// TIA Portal V18 export
FUNCTION_BLOCK "Aux_Motor_Control"   // FB12, LAD
{ S7_Optimized_Access := 'TRUE' }
// Written BY Kristopher Gimenez January 25,2023
// This block is used to control the Aux, and Cooler fan motors.
// stored: AutoNumber false, MemoryReserve 100, SetENOAutomatically false
   VAR
      AuxPumpStartTOF { S7_SetPoint := 'True'} : TOF_TIME;
      AuxPumpFailTON { S7_SetPoint := 'True'} : TON_TIME;
      CoolingFanFailTON { S7_SetPoint := 'True'} : TON_TIME;
      CoolingFanStartTON { S7_SetPoint := 'True'} : TOF_TIME;
   END_VAR
BEGIN

REGION Network 1: Aux Pump Start
   // TOFF used on Aux pump allows 2 seconds for functions to stop when system is disabled before pump is shutdown and to maintain while switching between Aux and TD Enabled
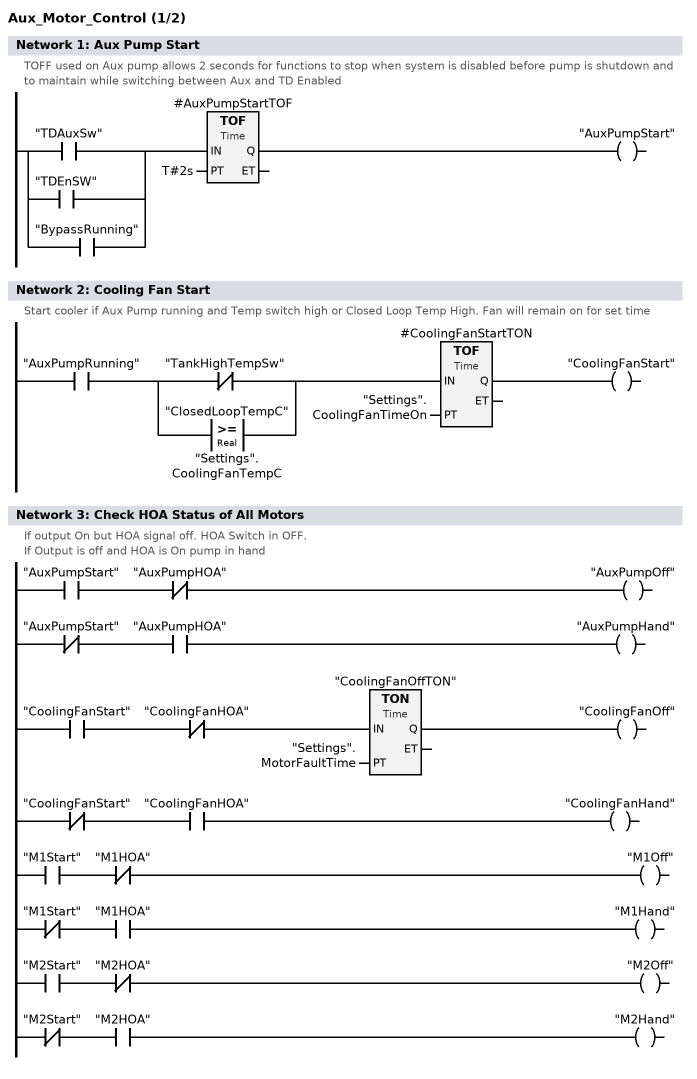
   RUNG wire#powerrail
      Contact( "TDAuxSw" )
      wire#w1
      { S7_Templates := "time_type := Time" } #AuxPumpStartTOF.TOF(pt := T#2s, et =>)
      Coil( "AuxPumpStart" )
   END_RUNG
   RUNG wire#powerrail
      Contact( "TDEnSW" )
   END_RUNG wire#w1
   RUNG wire#powerrail
      Contact( "BypassRunning" )
   END_RUNG wire#w1
   // the same network as SCL:
   #AuxPumpStartTOF(IN := "TDAuxSw" OR "TDEnSW" OR "BypassRunning", PT := T#2s);   // TOF
   "AuxPumpStart" := #AuxPumpStartTOF.Q;
END_REGION

REGION Network 2: Cooling Fan Start
   // Start cooler if Aux Pump running and Temp switch high or Closed Loop Temp High. Fan will remain on for set time
   RUNG wire#powerrail
      Contact( "AuxPumpRunning" )
      wire#w1
      I_Contact( "TankHighTempSw" )
      wire#w2
      { S7_Templates := "time_type := Time" } #CoolingFanStartTON.TOF(pt := "Settings".CoolingFanTimeOn, et =>)
      Coil( "CoolingFanStart" )
   END_RUNG
   RUNG wire#w1
      { S7_Templates := "SrcType := Real" } GE_Contact(in1 := "ClosedLoopTempC", in2 := "Settings".CoolingFanTempC)
   END_RUNG wire#w2
   // the same network as SCL:
   #CoolingFanStartTON(IN := "AuxPumpRunning" AND (NOT "TankHighTempSw" OR ("ClosedLoopTempC" >= "Settings".CoolingFanTempC)),   // TOF
                       PT := "Settings".CoolingFanTimeOn);
   "CoolingFanStart" := #CoolingFanStartTON.Q;
END_REGION

REGION Network 3: Check HOA Status of All Motors
   // If output On but HOA signal off. HOA Switch in OFF. 
   // If Output is off and HOA is On pump in hand
   RUNG wire#powerrail
      Contact( "AuxPumpStart" )
      I_Contact( "AuxPumpHOA" )
      Coil( "AuxPumpOff" )
   END_RUNG
   RUNG wire#powerrail
      I_Contact( "AuxPumpStart" )
      Contact( "AuxPumpHOA" )
      Coil( "AuxPumpHand" )
   END_RUNG
   RUNG wire#powerrail
      Contact( "CoolingFanStart" )
      I_Contact( "CoolingFanHOA" )
      { S7_Templates := "time_type := Time" } "CoolingFanOffTON".TON(pt := "Settings".MotorFaultTime, et =>)
      Coil( "CoolingFanOff" )
   END_RUNG
   RUNG wire#powerrail
      I_Contact( "CoolingFanStart" )
      Contact( "CoolingFanHOA" )
      Coil( "CoolingFanHand" )
   END_RUNG
   RUNG wire#powerrail
      Contact( "M1Start" )
      I_Contact( "M1HOA" )
      Coil( "M1Off" )
   END_RUNG
   RUNG wire#powerrail
      I_Contact( "M1Start" )
      Contact( "M1HOA" )
      Coil( "M1Hand" )
   END_RUNG
   RUNG wire#powerrail
      Contact( "M2Start" )
      I_Contact( "M2HOA" )
      Coil( "M2Off" )
   END_RUNG
   RUNG wire#powerrail
      I_Contact( "M2Start" )
      Contact( "M2HOA" )
      Coil( "M2Hand" )
   END_RUNG
   // the same network as SCL:
   "AuxPumpOff" := "AuxPumpStart" AND NOT "AuxPumpHOA";
   "AuxPumpHand" := NOT "AuxPumpStart" AND "AuxPumpHOA";
   "CoolingFanOffTON".TON(IN := "CoolingFanStart" AND NOT "CoolingFanHOA", PT := "Settings".MotorFaultTime);
   "CoolingFanOff" := "CoolingFanOffTON".Q;
   "CoolingFanHand" := NOT "CoolingFanStart" AND "CoolingFanHOA";
   "M1Off" := "M1Start" AND NOT "M1HOA";
   "M1Hand" := NOT "M1Start" AND "M1HOA";
   "M2Off" := "M2Start" AND NOT "M2HOA";
   "M2Hand" := NOT "M2Start" AND "M2HOA";
END_REGION

REGION Network 4: Motor Starter Fault Status
   // If pump start signal seen on HOA input but it has not started by fault time. Set motor fault
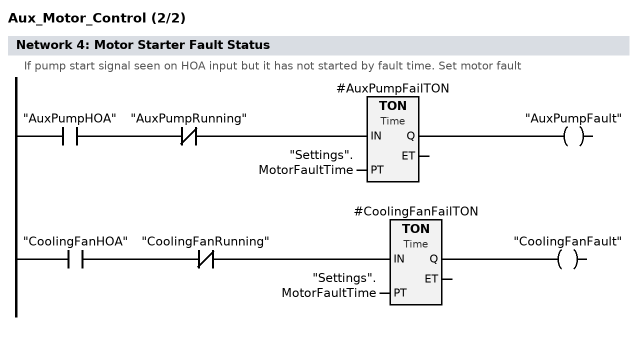
   RUNG wire#powerrail
      Contact( "AuxPumpHOA" )
      I_Contact( "AuxPumpRunning" )
      { S7_Templates := "time_type := Time" } #AuxPumpFailTON.TON(pt := "Settings".MotorFaultTime, et =>)
      Coil( "AuxPumpFault" )
   END_RUNG
   RUNG wire#powerrail
      Contact( "CoolingFanHOA" )
      I_Contact( "CoolingFanRunning" )
      { S7_Templates := "time_type := Time" } #CoolingFanFailTON.TON(pt := "Settings".MotorFaultTime, et =>)
      Coil( "CoolingFanFault" )
   END_RUNG
   // the same network as SCL:
   #AuxPumpFailTON(IN := "AuxPumpHOA" AND NOT "AuxPumpRunning", PT := "Settings".MotorFaultTime);   // TON
   "AuxPumpFault" := #AuxPumpFailTON.Q;
   #CoolingFanFailTON(IN := "CoolingFanHOA" AND NOT "CoolingFanRunning", PT := "Settings".MotorFaultTime);   // TON
   "CoolingFanFault" := #CoolingFanFailTON.Q;
END_REGION
END_FUNCTION_BLOCK
